(*
version 1.0	26. oct. 2008
programmer 	hugo
tested by		tobias

this function calculates the Cauchy distribution function

*)
FUNCTION CAUCHYCD : REAL
VAR_INPUT
	X : REAL;
	T : REAL;
	U : REAL;
END_VAR

CAUCHYCD := 0.5 + math.PI_INV * ATAN((X - T) / U);



(* revision hisdtory
hm	26. oct. 2008	rev 1.0
	original version

*)

END_FUNCTION

(* stored: Version 1.1.0.1
   POU CAUCHYCD: Id {7d7c77dd-bc1f-4d41-adad-7c0f488b7664}, SpecialFunc None *)
